FUNCTION_BLOCK FB_Quaternion IMPLEMENTS I_Quat
VAR
    fw : LREAL;
    fx : LREAL;
    fy : LREAL;
    fz : LREAL;
END_VAR


METHOD AddQuat
VAR_INPUT
    iQuat	: I_Quat;
END_VAR

w := w + iQuat.w;
x := x + iQuat.x;
y := y + iQuat.y;
z := z + iQuat.z;
END_METHOD


METHOD DivQuat
VAR_INPUT
    iQuat	: I_Quat;
END_VAR
VAR_OUTPUT
    bError : BOOL;
    sErrorMsg : T_MaxString;
END_VAR
VAR
    fNormSq : LREAL;
    fwi : LREAL;
    fxi : LREAL;
    fyi : LREAL;
    fzi : LREAL;
END_VAR

bError := FALSE;
sErrorMsg := '';

fNormSq := F_NormSqQuat(iQuat);

IF fNormSq = 0.0 THEN
    bError := TRUE;
    sErrorMsg := 'Error: cannot divide by a quaternion with a norm of 0.';
    RETURN;
END_IF

fwi := w;
fxi := x;
fyi := y;
fzi := z;

w := ((iQuat.w * fwi) + (iQuat.x * fxi) + (iQuat.y * fyi) + (iQuat.z * fzi)) / fNormSq;
x := ((iQuat.w * fxi) - (iQuat.x * fwi) - (iQuat.y * fzi) + (iQuat.z * fyi)) / fNormSq;
y := ((iQuat.w * fyi) + (iQuat.x * fzi) - (iQuat.y * fwi) - (iQuat.z * fxi)) / fNormSq;
z := ((iQuat.w * fzi) - (iQuat.x * fyi) + (iQuat.y * fxi) - (iQuat.z * fwi)) / fNormSq;
END_METHOD


METHOD DivScalar
VAR_INPUT
    fScalar : LREAL;
END_VAR
VAR_OUTPUT
    bError : BOOL;
    sErrorMsg : T_MaxString;
END_VAR

bError := FALSE;
sErrorMsg := '';

IF fScalar = 0.0 THEN
    bError := TRUE;
    sErrorMsg := 'Error: attempted division of quaternion by scalar of 0.';
    RETURN;
END_IF

w := w / fScalar;
x := x / fScalar;
y := y / fScalar;
z := z / fScalar;
END_METHOD


METHOD EqualsQuat : BOOL
VAR_INPUT
    iQuat	: I_Quat;
END_VAR

EqualsQuat := w = iQuat.w AND
              x = iQuat.x AND
              y = iQuat.y AND
              z = iQuat.z;
END_METHOD


METHOD GetNorm : LREAL

GetNorm := SQRT(w*w + x*x + y*y + z*z);
END_METHOD


METHOD GetNormSq : LREAL

GetNormSq := w*w + x*x + y*y + z*z;
END_METHOD


METHOD MakeConj

w := w;
x := -x;
y := -y;
z := -z;
END_METHOD


METHOD MulQuat
VAR_INPUT
    iQuat	: I_Quat;
END_VAR
VAR
    fwi : LREAL;
    fxi : LREAL;
    fyi : LREAL;
    fzi : LREAL;
END_VAR

fwi := w;
fxi := x;
fyi := y;
fzi := z;

w := (fwi * iQuat.w) - (fxi * iQuat.x) - (fyi * iQuat.y) - (fzi * iQuat.z);
x := (fwi * iQuat.x) + (fxi * iQuat.w) + (fyi * iQuat.z) - (fzi * iQuat.y);
y := (fwi * iQuat.y) - (fxi * iQuat.z) + (fyi * iQuat.w) + (fzi * iQuat.x);
z := (fwi * iQuat.z) + (fxi * iQuat.y) - (fyi * iQuat.x) + (fzi * iQuat.w);
END_METHOD


METHOD Normalize
VAR_OUTPUT
    bError : BOOL;
    sErrorMsg : T_MaxString;
END_VAR
VAR
    fNorm : LREAL;
END_VAR

bError := FALSE;
sErrorMsg := '';

fNorm := GetNorm();

IF fNorm = 0.0 THEN
    bError := TRUE;
    sErrorMsg := 'Error: cannot normalize a quaternion with a norm of 0.';
    RETURN;
END_IF

w := w / fNorm;
x := x / fNorm;
y := y / fNorm;
z := z / fNorm;
END_METHOD


METHOD Set
VAR_INPUT
    w : LREAL;
    i : LREAL;
    j : LREAL;
    k : LREAL;
END_VAR

THIS^.w := w;
THIS^.x := i;
THIS^.y := j;
THIS^.z := k;
END_METHOD


METHOD ToString : T_MaxString

ToString := '';

IF w < 0.0 THEN
    ToString := CONCAT(ToString, '-');
END_IF

ToString := CONCAT(ToString, LREAL_TO_STRING(ABS(w)));

IF x >= 0.0 THEN
    ToString := CONCAT(ToString, ' + ');
ELSE
    ToString := CONCAT(ToString, ' - ');
END_IF

ToString := CONCAT(ToString, LREAL_TO_STRING(ABS(x)));
ToString := CONCAT(ToString, 'i');

IF y >= 0.0 THEN
    ToString := CONCAT(ToString, ' + ');
ELSE
    ToString := CONCAT(ToString, ' - ');
END_IF

ToString := CONCAT(ToString, LREAL_TO_STRING(ABS(y)));
ToString := CONCAT(ToString, 'j');

IF z >= 0.0 THEN
    ToString := CONCAT(ToString, ' + ');
ELSE
    ToString := CONCAT(ToString, ' - ');
END_IF

ToString := CONCAT(ToString, LREAL_TO_STRING(ABS(z)));
ToString := CONCAT(ToString, 'k');
END_METHOD


PROPERTY w : LREAL
GET

w := fw;
END_GET
SET

fw := w;
END_SET
END_PROPERTY


PROPERTY x : LREAL
GET

x := fx;
END_GET
SET

fx := x;
END_SET
END_PROPERTY


PROPERTY y : LREAL
GET

y := fy;
END_GET
SET

fy := y;
END_SET
END_PROPERTY


PROPERTY z : LREAL
GET

z := fz;
END_GET
SET

fz := z;
END_SET
END_PROPERTY

END_FUNCTION_BLOCK

(* stored: Version 1.1.0.1
   POU FB_Quaternion: Id {368e3e81-21d8-4842-8003-27045a72af0c}, SpecialFunc None
   Method AddQuat: Id {f9d2f632-88d1-43c0-b869-4c86af2cc83c}
   Method DivQuat: Id {1915c45d-0c4c-4cb5-9348-b641b28e4fe4}
   Method DivScalar: Id {4d84e2f2-81a3-414a-b1e8-9a34fadfe7d1}
   Method EqualsQuat: Id {b2ebfb21-208a-4535-9c1d-8fb4ad4e160f}
   Method GetNorm: Id {172c3d10-6a52-4e90-853d-ef52c393f88d}
   Method GetNormSq: Id {f4b27ab1-ff46-4a03-8e7e-5b8182f21d26}
   Method MakeConj: Id {0d0a6a03-d7f4-464e-b9c6-f4816551c4f1}
   Method MulQuat: Id {6c286bdd-7e84-46da-8460-b9d9c214f657}
   Method Normalize: Id {eb8f3894-180f-4c3d-b1a9-a26e4a1164ab}
   Method Set: Id {0fe647d3-f4aa-4086-b995-65bfafb09ef8}
   Method ToString: Id {54f42700-7127-410c-be09-fde5d937a7ae}
   Property w: Id {17f98bc7-9353-4a99-8e24-cb6cc3bff018}
   Get Get: Id {f87b7f71-d6b3-4a5e-82b9-7aed2063a787}
   Set Set: Id {514f658b-9130-4171-89fa-63e9f5da998b}
   Property x: Id {9f7d7ec1-ea69-4a4d-ad05-ebda0a502293}
   Get Get: Id {34c5f1f9-74e6-49d2-84bf-38d7a7580d8b}
   Set Set: Id {c7bb6447-2983-4e5a-b29b-7714cd2126d7}
   Property y: Id {4c760f40-696a-4501-848e-c0bb02a44ff6}
   Get Get: Id {fb4ee227-0c91-40b0-995d-11d7d79c23c2}
   Set Set: Id {594c8029-8ed6-4e20-8454-fdc93c7b80c8}
   Property z: Id {93a01f3f-5090-43d2-b56a-8cd7586ad31c}
   Get Get: Id {b3c22bdd-55c2-483c-810f-ea1fc45d6b7d}
   Set Set: Id {e1a56b12-5ba1-4ab1-84ca-a2b2af0ceeab} *)
